% RSLogix 500 project ALSAFE.RSS, saved by version 8.10.00.18 %
PROJECT "ALSAFE"    % processor: SLC 500, 1747-L542 %

PROGRAM FILES
  LAD 2   73 rungs
  LAD 3   98 rungs
  LAD 4   40 rungs
  LAD 5   5 rungs
  LAD 6   89 rungs
  LAD 9   48 rungs
  LAD 10   101 rungs
  LAD 11   76 rungs
  LAD 15   61 rungs
  LAD 16   10 rungs
  LAD 17   20 rungs
  LAD 21   5 rungs
  LAD 22   77 rungs
  LAD 25   112 rungs
  LAD 26   32 rungs
  LAD 27   42 rungs
  LAD 30   28 rungs
  LAD 31   116 rungs
  LAD 32   20 rungs
  LAD 40   35 rungs
  LAD 50   183 rungs
  LAD 51   113 rungs
  LAD 52   5 rungs
  LAD 53   5 rungs
  LAD 71   9 rungs
  LAD 75   15 rungs
  LAD 76   23 rungs
  LAD 77   4 rungs
  LAD 78   4 rungs
  LAD 80   11 rungs

DATA FILES
  O0 OUTPUT  20 elements
  I1 INPUT  19 elements
  S2 STATUS  164 elements
  B3 BINARY  68 elements
  T4 TIMER  32 elements
  C5 COUNTER  2 elements
  R6 CONTROL  12 elements
  N7 INTEGER  131 elements
  F8 FLOAT  15 elements
  N9   25 elements
  B10   110 elements
  B11   63 elements
  T13   10 elements
  B15   1 elements
  B16   20 elements
  B17   28 elements
  T21   65 elements
  B22   11 elements
  B23   4 elements
  N25   210 elements
  B29   12 elements
  T31   40 elements
  N32   14 elements
  N40   60 elements
  N41   60 elements
  N42   120 elements
  B49   2 elements
  N50   54 elements
  N51   210 elements
  N52   18 elements
  B53   100 elements
  N54   31 elements
  N60   54 elements
  N75   250 elements
  N76   100 elements
  N90   5 elements
  N91   250 elements
  N92   250 elements
  N100   101 elements
  N104   12 elements
  N105   102 elements
  N106   1 elements
  N107   27 elements
  N108   12 elements
  N109   31 elements
  N111   214 elements

LADDER 2
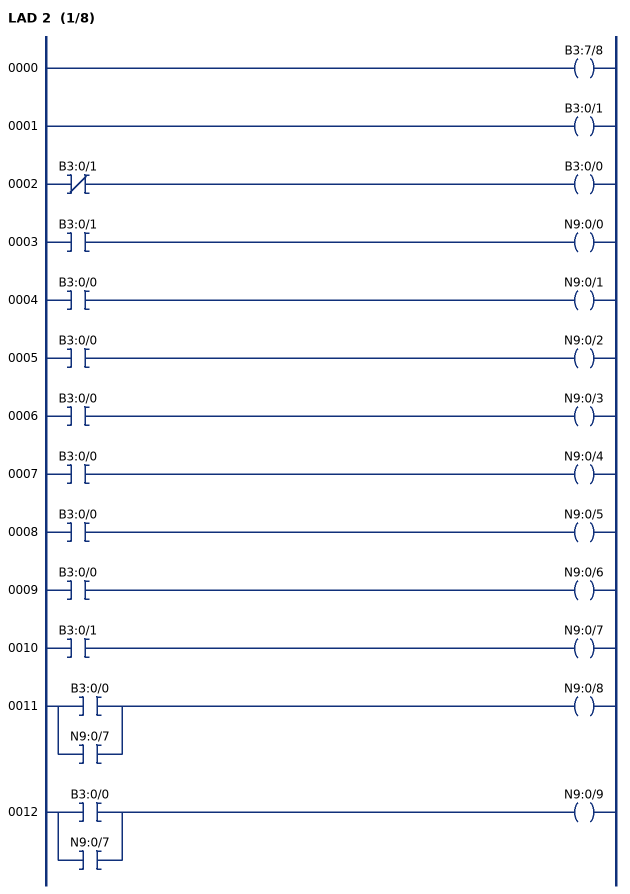
% Rung: 0 %
SOR OTE B3:7/8 EOR
% Rung: 1 %
SOR OTE B3:0/1 EOR
% Rung: 2 %
SOR XIO B3:0/1 OTE B3:0/0 EOR
% Rung: 3 %
SOR XIC B3:0/1 OTE N9:0/0 EOR
% Rung: 4 %
SOR XIC B3:0/0 OTE N9:0/1 EOR
% Rung: 5 %
SOR XIC B3:0/0 OTE N9:0/2 EOR
% Rung: 6 %
SOR XIC B3:0/0 OTE N9:0/3 EOR
% Rung: 7 %
SOR XIC B3:0/0 OTE N9:0/4 EOR
% Rung: 8 %
SOR XIC B3:0/0 OTE N9:0/5 EOR
% Rung: 9 %
SOR XIC B3:0/0 OTE N9:0/6 EOR
% Rung: 10 %
SOR XIC B3:0/1 OTE N9:0/7 EOR
% Rung: 11 %
SOR BST XIC B3:0/0 NXB XIC N9:0/7 BND OTE N9:0/8 EOR
% Rung: 12 %
SOR BST XIC B3:0/0 NXB XIC N9:0/7 BND OTE N9:0/9 EOR

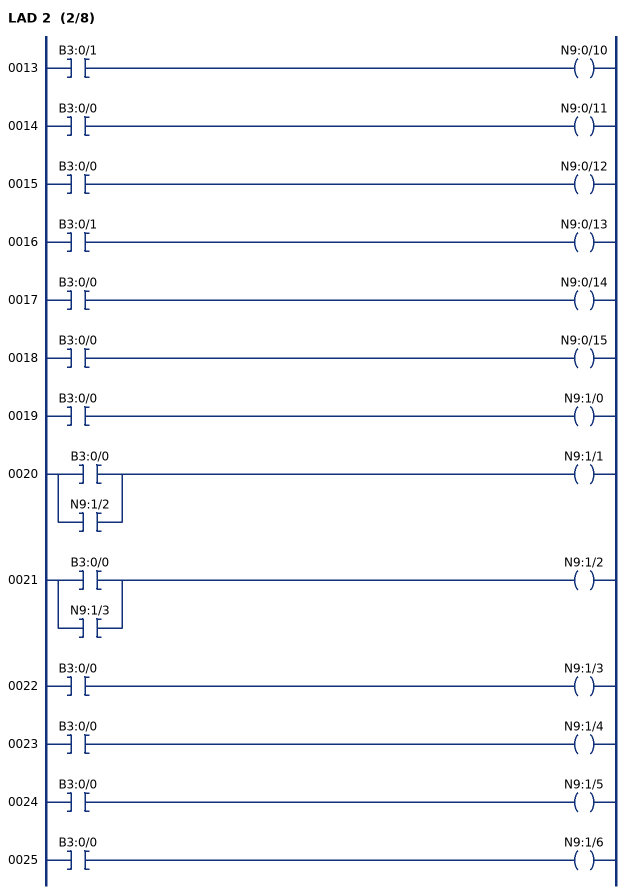
% Rung: 13 %
SOR XIC B3:0/1 OTE N9:0/10 EOR
% Rung: 14 %
SOR XIC B3:0/0 OTE N9:0/11 EOR
% Rung: 15 %
SOR XIC B3:0/0 OTE N9:0/12 EOR
% Rung: 16 %
SOR XIC B3:0/1 OTE N9:0/13 EOR
% Rung: 17 %
SOR XIC B3:0/0 OTE N9:0/14 EOR
% Rung: 18 %
SOR XIC B3:0/0 OTE N9:0/15 EOR
% Rung: 19 %
SOR XIC B3:0/0 OTE N9:1/0 EOR
% Rung: 20 %
SOR BST XIC B3:0/0 NXB XIC N9:1/2 BND OTE N9:1/1 EOR
% Rung: 21 %
SOR BST XIC B3:0/0 NXB XIC N9:1/3 BND OTE N9:1/2 EOR
% Rung: 22 %
SOR XIC B3:0/0 OTE N9:1/3 EOR
% Rung: 23 %
SOR XIC B3:0/0 OTE N9:1/4 EOR
% Rung: 24 %
SOR XIC B3:0/0 OTE N9:1/5 EOR
% Rung: 25 %
SOR XIC B3:0/0 OTE N9:1/6 EOR

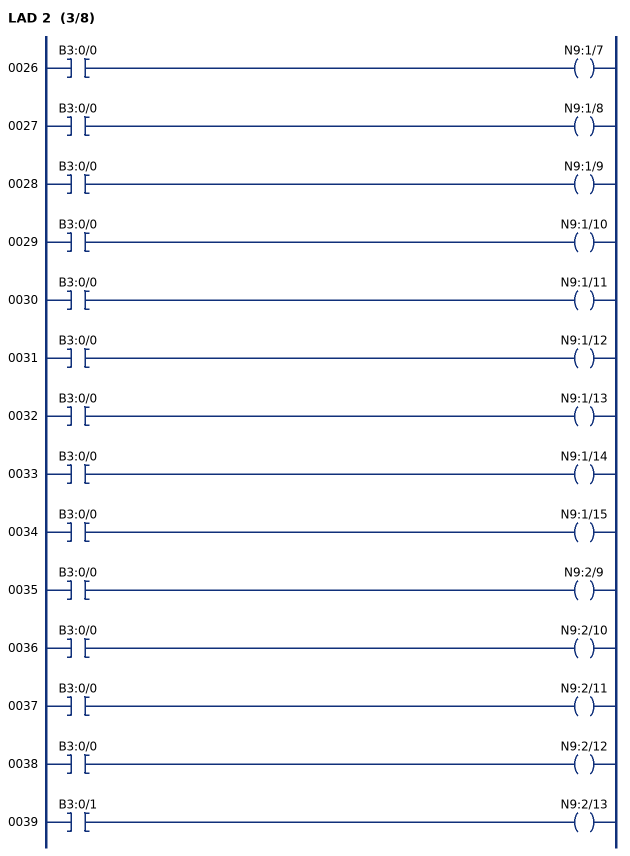
% Rung: 26 %
SOR XIC B3:0/0 OTE N9:1/7 EOR
% Rung: 27 %
SOR XIC B3:0/0 OTE N9:1/8 EOR
% Rung: 28 %
SOR XIC B3:0/0 OTE N9:1/9 EOR
% Rung: 29 %
SOR XIC B3:0/0 OTE N9:1/10 EOR
% Rung: 30 %
SOR XIC B3:0/0 OTE N9:1/11 EOR
% Rung: 31 %
SOR XIC B3:0/0 OTE N9:1/12 EOR
% Rung: 32 %
SOR XIC B3:0/0 OTE N9:1/13 EOR
% Rung: 33 %
SOR XIC B3:0/0 OTE N9:1/14 EOR
% Rung: 34 %
SOR XIC B3:0/0 OTE N9:1/15 EOR
% Rung: 35 %
SOR XIC B3:0/0 OTE N9:2/9 EOR
% Rung: 36 %
SOR XIC B3:0/0 OTE N9:2/10 EOR
% Rung: 37 %
SOR XIC B3:0/0 OTE N9:2/11 EOR
% Rung: 38 %
SOR XIC B3:0/0 OTE N9:2/12 EOR
% Rung: 39 %
SOR XIC B3:0/1 OTE N9:2/13 EOR

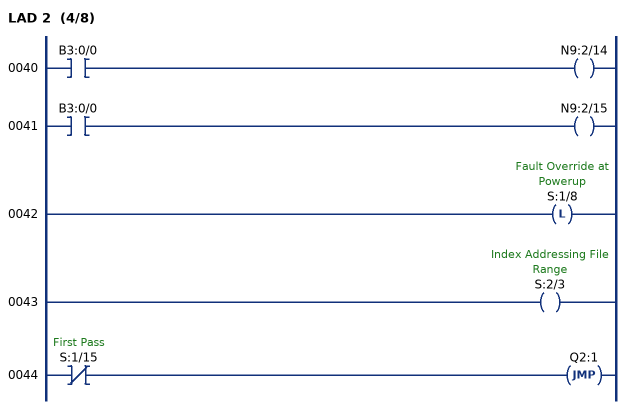
% Rung: 40 %
SOR XIC B3:0/0 OTE N9:2/14 EOR
% Rung: 41 %
SOR XIC B3:0/0 OTE N9:2/15 EOR
% Rung: 42 %
SOR OTL S:1/8 EOR
%   S:1/8  "Fault Override at Powerup" %
% Rung: 43 %
SOR OTE S:2/3 EOR
%   S:2/3  "Index Addressing File Range" %
% Rung: 44 %
SOR XIO S:1/15 JMP Q2:1 EOR
%   S:1/15  "First Pass" %

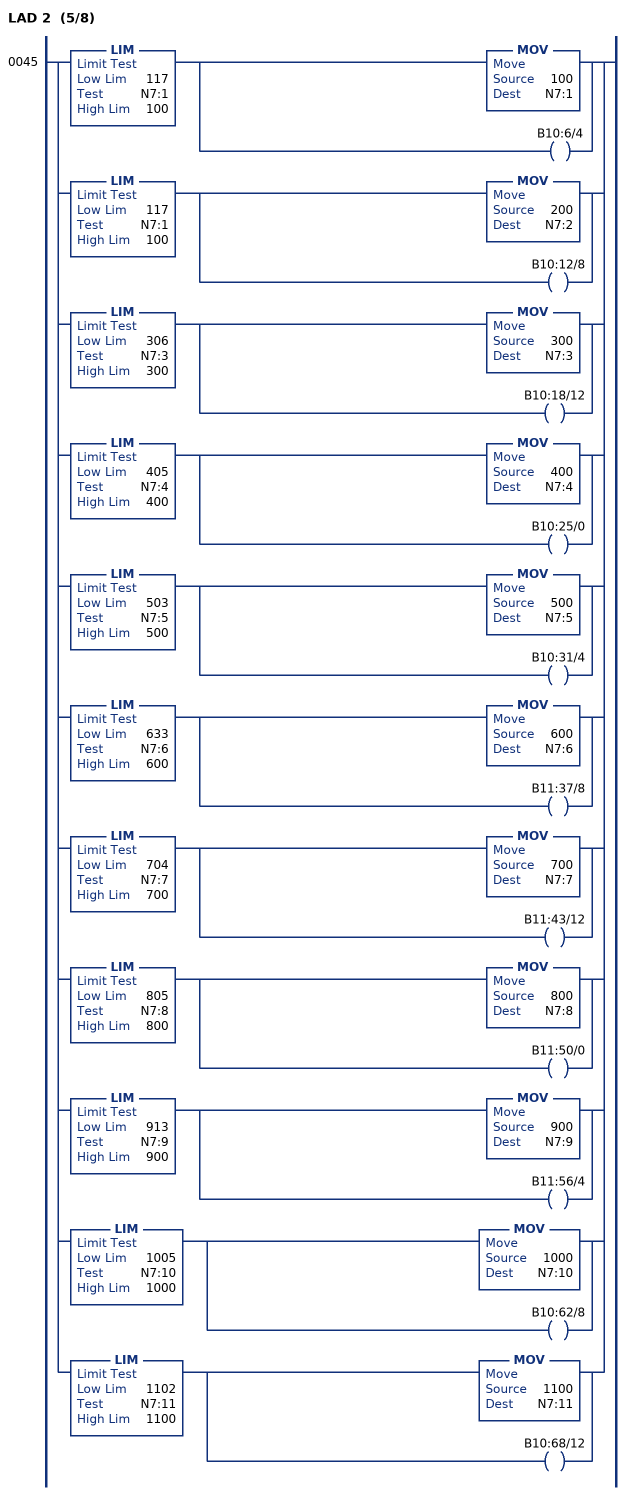
% Rung: 45 %
SOR BST LIM 117 N7:1 100 BST MOV 100 N7:1 NXB OTE B10:6/4 BND NXB LIM 117 N7:1 100 BST MOV 200 N7:2 NXB OTE B10:12/8 BND NXB LIM 306 N7:3 300 BST MOV 300 N7:3 NXB OTE B10:18/12 BND NXB LIM 405 N7:4 400 BST MOV 400 N7:4 NXB OTE B10:25/0 BND NXB LIM 503 N7:5 500 BST MOV 500 N7:5 NXB OTE B10:31/4 BND NXB LIM 633 N7:6 600 BST MOV 600 N7:6 NXB OTE B11:37/8 BND NXB LIM 704 N7:7 700 BST MOV 700 N7:7 NXB OTE B11:43/12 BND NXB LIM 805 N7:8 800 BST MOV 800 N7:8 NXB OTE B11:50/0 BND NXB LIM 913 N7:9 900 BST MOV 900 N7:9 NXB OTE B11:56/4 BND NXB LIM 1005 N7:10 1000 BST MOV 1000 N7:10 NXB OTE B10:62/8 BND NXB LIM 1102 N7:11 1100 BST MOV 1100 N7:11 NXB OTE B10:68/12 BND BND EOR

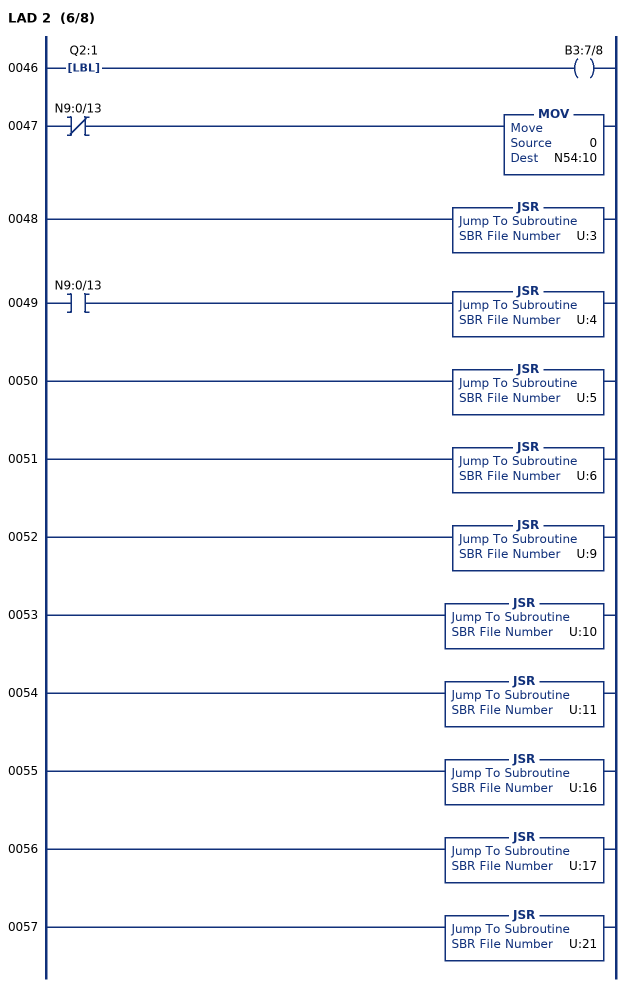
% Rung: 46 %
SOR LBL Q2:1 OTE B3:7/8 EOR
% Rung: 47 %
SOR XIO N9:0/13 MOV 0 N54:10 EOR
% Rung: 48 %
SOR JSR U:3 EOR
% Rung: 49 %
SOR XIC N9:0/13 JSR U:4 EOR
% Rung: 50 %
SOR JSR U:5 EOR
% Rung: 51 %
SOR JSR U:6 EOR
% Rung: 52 %
SOR JSR U:9 EOR
% Rung: 53 %
SOR JSR U:10 EOR
% Rung: 54 %
SOR JSR U:11 EOR
% Rung: 55 %
SOR JSR U:16 EOR
% Rung: 56 %
SOR JSR U:17 EOR
% Rung: 57 %
SOR JSR U:21 EOR

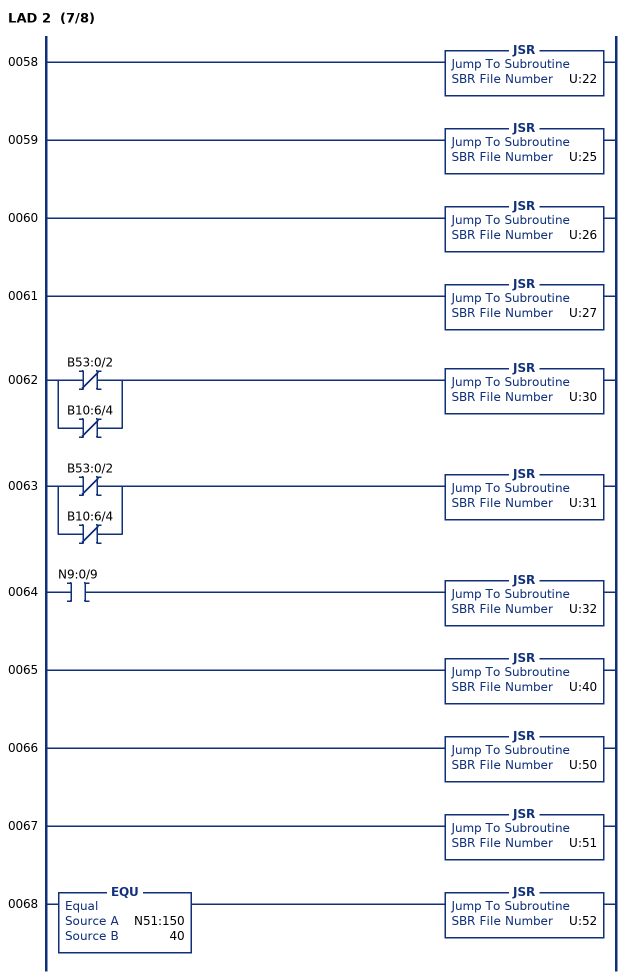
% Rung: 58 %
SOR JSR U:22 EOR
% Rung: 59 %
SOR JSR U:25 EOR
% Rung: 60 %
SOR JSR U:26 EOR
% Rung: 61 %
SOR JSR U:27 EOR
% Rung: 62 %
SOR BST XIO B53:0/2 NXB XIO B10:6/4 BND JSR U:30 EOR
% Rung: 63 %
SOR BST XIO B53:0/2 NXB XIO B10:6/4 BND JSR U:31 EOR
% Rung: 64 %
SOR XIC N9:0/9 JSR U:32 EOR
% Rung: 65 %
SOR JSR U:40 EOR
% Rung: 66 %
SOR JSR U:50 EOR
% Rung: 67 %
SOR JSR U:51 EOR
% Rung: 68 %
SOR EQU N51:150 40 JSR U:52 EOR

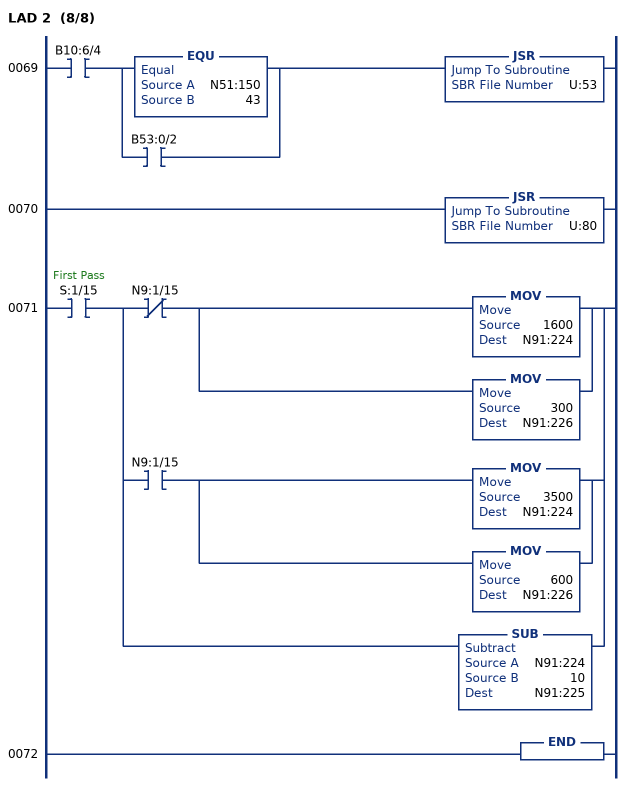
% Rung: 69 %
SOR XIC B10:6/4 BST EQU N51:150 43 NXB XIC B53:0/2 BND JSR U:53 EOR
% Rung: 70 %
SOR JSR U:80 EOR
% Rung: 71 %
SOR XIC S:1/15 BST XIO N9:1/15 BST MOV 1600 N91:224 NXB MOV 300 N91:226 BND NXB XIC N9:1/15 BST MOV 3500 N91:224 NXB MOV 600 N91:226 BND NXB SUB N91:224 10 N91:225 BND EOR
%   S:1/15  "First Pass" %
% Rung: 72 %
SOR END EOR

LADDER 3
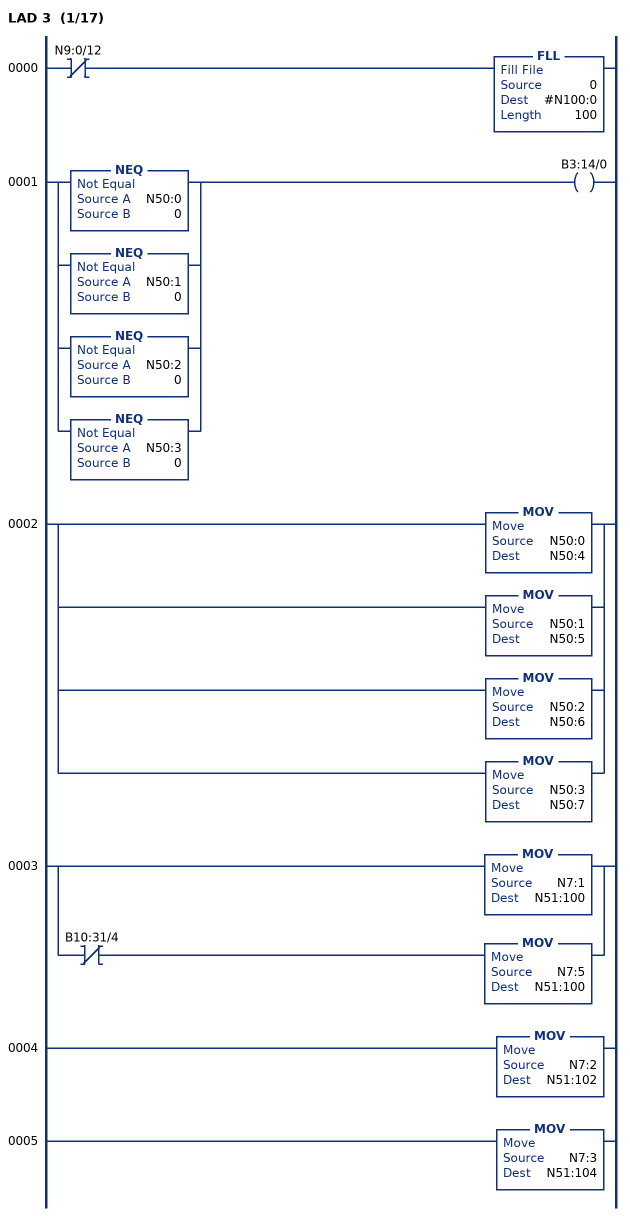
% Rung: 0 %
SOR XIO N9:0/12 FLL 0 #N100:0 100 EOR
% Rung: 1 %
SOR BST NEQ N50:0 0 NXB NEQ N50:1 0 NXB NEQ N50:2 0 NXB NEQ N50:3 0 BND OTE B3:14/0 EOR
% Rung: 2 %
SOR BST MOV N50:0 N50:4 NXB MOV N50:1 N50:5 NXB MOV N50:2 N50:6 NXB MOV N50:3 N50:7 BND EOR
% Rung: 3 %
SOR BST MOV N7:1 N51:100 NXB XIO B10:31/4 MOV N7:5 N51:100 BND EOR
% Rung: 4 %
SOR MOV N7:2 N51:102 EOR
% Rung: 5 %
SOR MOV N7:3 N51:104 EOR

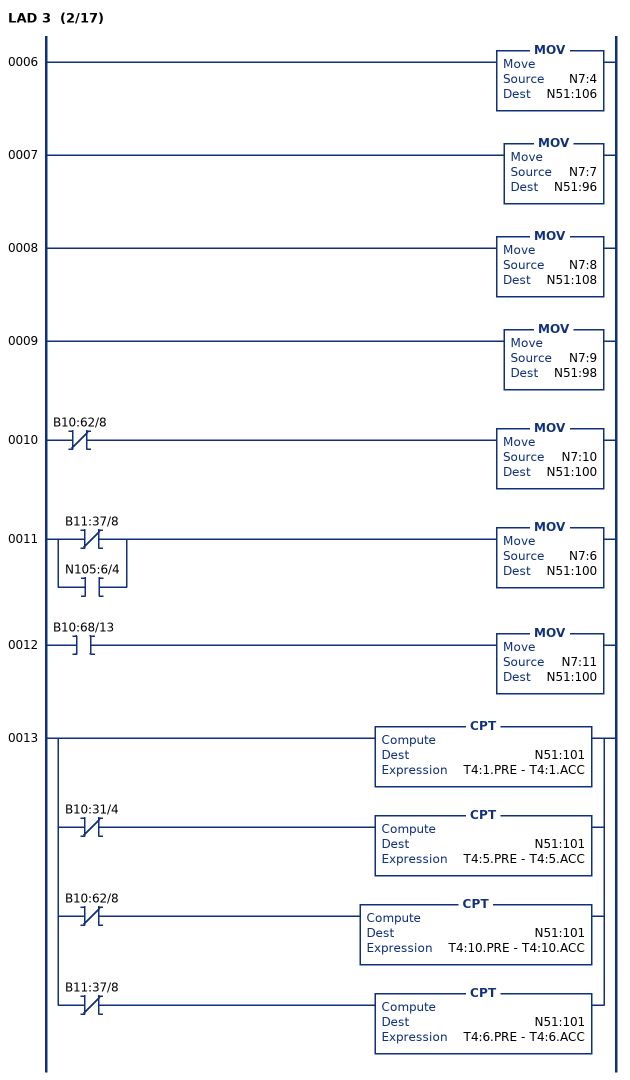
% Rung: 6 %
SOR MOV N7:4 N51:106 EOR
% Rung: 7 %
SOR MOV N7:7 N51:96 EOR
% Rung: 8 %
SOR MOV N7:8 N51:108 EOR
% Rung: 9 %
SOR MOV N7:9 N51:98 EOR
% Rung: 10 %
SOR XIO B10:62/8 MOV N7:10 N51:100 EOR
% Rung: 11 %
SOR BST XIO B11:37/8 NXB XIC N105:6/4 BND MOV N7:6 N51:100 EOR
% Rung: 12 %
SOR XIC B10:68/13 MOV N7:11 N51:100 EOR
% Rung: 13 %
SOR BST CPT N51:101 " T4:1.PRE - T4:1.ACC " NXB XIO B10:31/4 CPT N51:101 " T4:5.PRE - T4:5.ACC " NXB XIO B10:62/8 CPT N51:101 " T4:10.PRE - T4:10.ACC " NXB XIO B11:37/8 CPT N51:101 " T4:6.PRE - T4:6.ACC " BND EOR

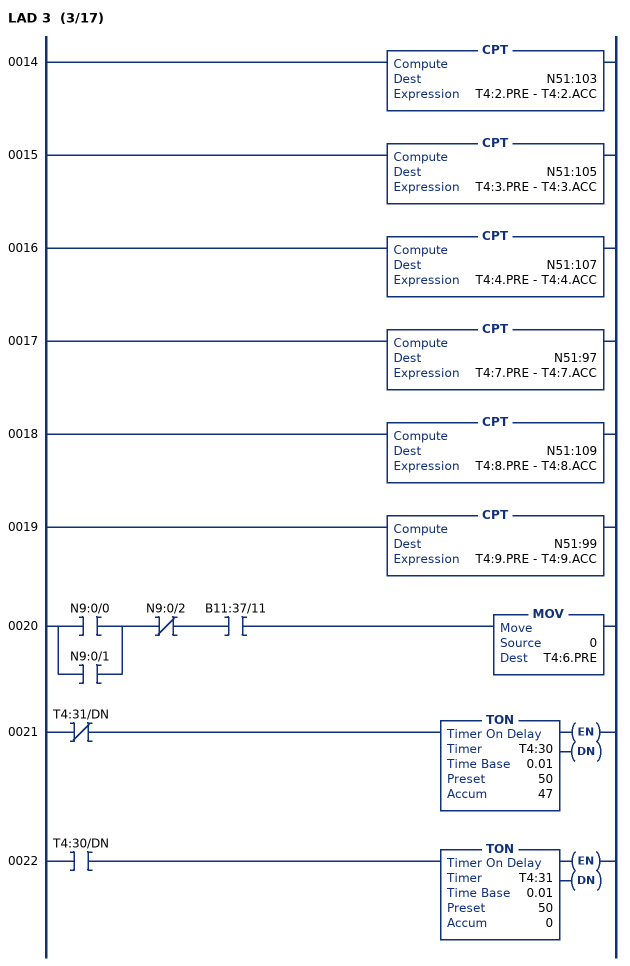
% Rung: 14 %
SOR CPT N51:103 " T4:2.PRE - T4:2.ACC " EOR
% Rung: 15 %
SOR CPT N51:105 " T4:3.PRE - T4:3.ACC " EOR
% Rung: 16 %
SOR CPT N51:107 " T4:4.PRE - T4:4.ACC " EOR
% Rung: 17 %
SOR CPT N51:97 " T4:7.PRE - T4:7.ACC " EOR
% Rung: 18 %
SOR CPT N51:109 " T4:8.PRE - T4:8.ACC " EOR
% Rung: 19 %
SOR CPT N51:99 " T4:9.PRE - T4:9.ACC " EOR
% Rung: 20 %
SOR BST XIC N9:0/0 NXB XIC N9:0/1 BND XIO N9:0/2 XIC B11:37/11 MOV 0 T4:6.PRE EOR
% Rung: 21 %
SOR XIO T4:31/DN TON T4:30 0.01 50 47 EOR
% Rung: 22 %
SOR XIC T4:30/DN TON T4:31 0.01 50 0 EOR

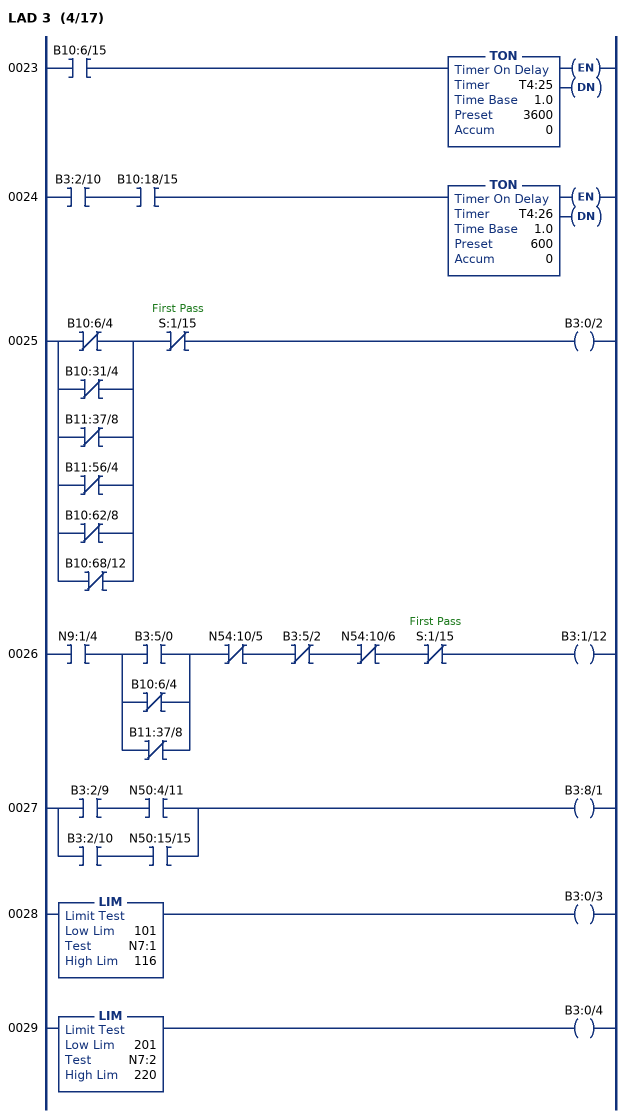
% Rung: 23 %
SOR XIC B10:6/15 TON T4:25 1.0 3600 0 EOR
% Rung: 24 %
SOR XIC B3:2/10 XIC B10:18/15 TON T4:26 1.0 600 0 EOR
% Rung: 25 %
SOR BST XIO B10:6/4 NXB XIO B10:31/4 NXB XIO B11:37/8 NXB XIO B11:56/4 NXB XIO B10:62/8 NXB XIO B10:68/12 BND XIO S:1/15 OTE B3:0/2 EOR
%   S:1/15  "First Pass" %
% Rung: 26 %
SOR XIC N9:1/4 BST XIC B3:5/0 NXB XIO B10:6/4 NXB XIO B11:37/8 BND XIO N54:10/5 XIO B3:5/2 XIO N54:10/6 XIO S:1/15 OTE B3:1/12 EOR
%   S:1/15  "First Pass" %
% Rung: 27 %
SOR BST XIC B3:2/9 XIC N50:4/11 NXB XIC B3:2/10 XIC N50:15/15 BND OTE B3:8/1 EOR
% Rung: 28 %
SOR LIM 101 N7:1 116 OTE B3:0/3 EOR
% Rung: 29 %
SOR LIM 201 N7:2 220 OTE B3:0/4 EOR

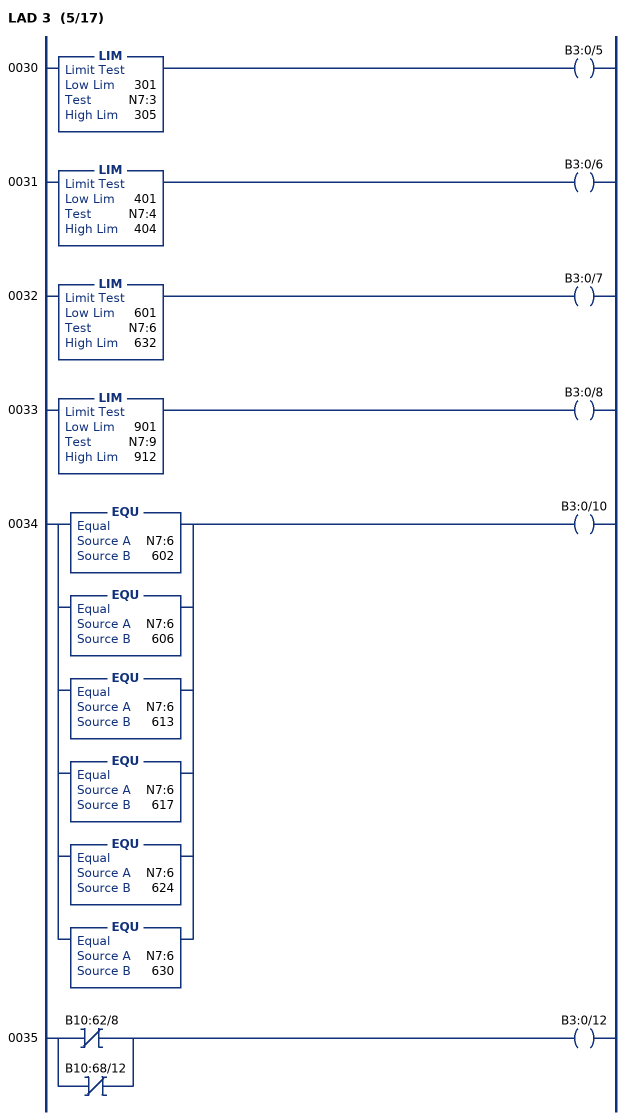
% Rung: 30 %
SOR LIM 301 N7:3 305 OTE B3:0/5 EOR
% Rung: 31 %
SOR LIM 401 N7:4 404 OTE B3:0/6 EOR
% Rung: 32 %
SOR LIM 601 N7:6 632 OTE B3:0/7 EOR
% Rung: 33 %
SOR LIM 901 N7:9 912 OTE B3:0/8 EOR
% Rung: 34 %
SOR BST EQU N7:6 602 NXB EQU N7:6 606 NXB EQU N7:6 613 NXB EQU N7:6 617 NXB EQU N7:6 624 NXB EQU N7:6 630 BND OTE B3:0/10 EOR
% Rung: 35 %
SOR BST XIO B10:62/8 NXB XIO B10:68/12 BND OTE B3:0/12 EOR

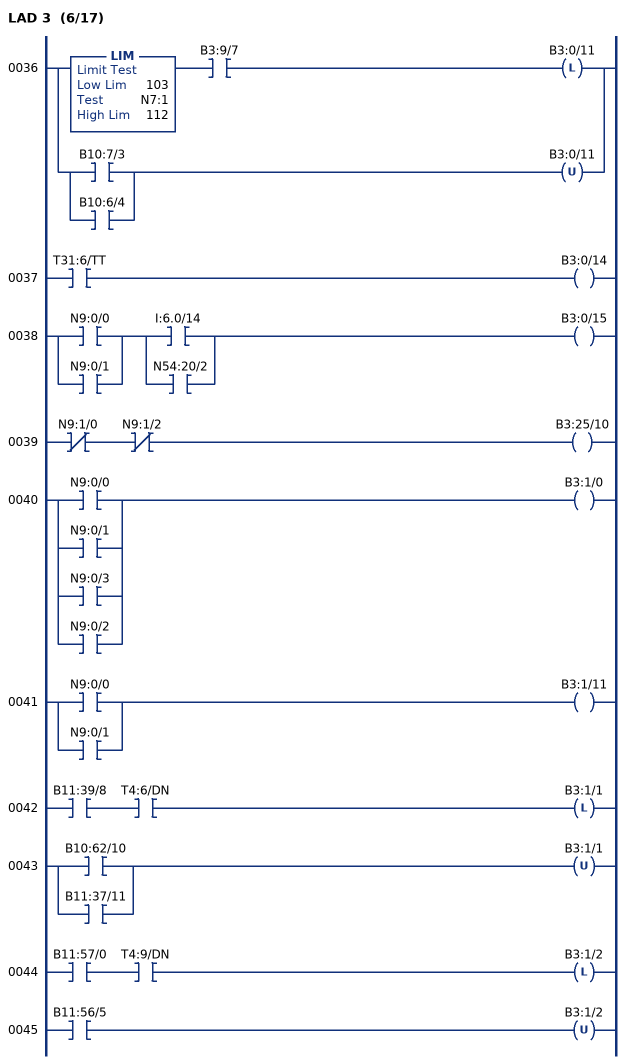
% Rung: 36 %
SOR BST LIM 103 N7:1 112 XIC B3:9/7 OTL B3:0/11 NXB BST XIC B10:7/3 NXB XIC B10:6/4 BND OTU B3:0/11 BND EOR
% Rung: 37 %
SOR XIC T31:6/TT OTE B3:0/14 EOR
% Rung: 38 %
SOR BST XIC N9:0/0 NXB XIC N9:0/1 BND BST XIC I:6.0/14 NXB XIC N54:20/2 BND OTE B3:0/15 EOR
% Rung: 39 %
SOR XIO N9:1/0 XIO N9:1/2 OTE B3:25/10 EOR
% Rung: 40 %
SOR BST XIC N9:0/0 NXB XIC N9:0/1 NXB XIC N9:0/3 NXB XIC N9:0/2 BND OTE B3:1/0 EOR
% Rung: 41 %
SOR BST XIC N9:0/0 NXB XIC N9:0/1 BND OTE B3:1/11 EOR
% Rung: 42 %
SOR XIC B11:39/8 XIC T4:6/DN OTL B3:1/1 EOR
% Rung: 43 %
SOR BST XIC B10:62/10 NXB XIC B11:37/11 BND OTU B3:1/1 EOR
% Rung: 44 %
SOR XIC B11:57/0 XIC T4:9/DN OTL B3:1/2 EOR
% Rung: 45 %
SOR XIC B11:56/5 OTU B3:1/2 EOR

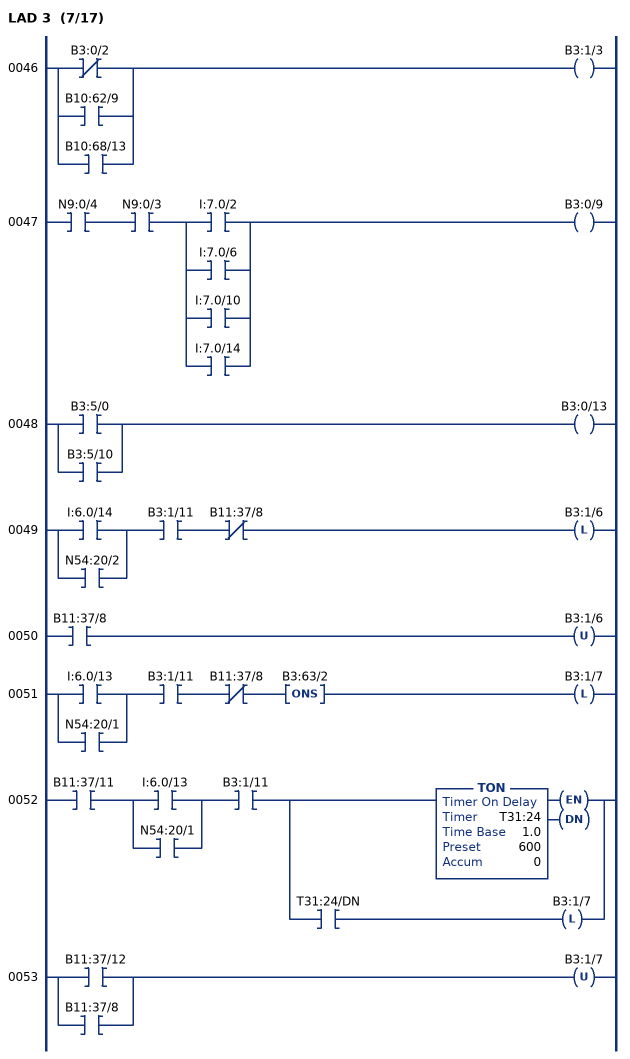
% Rung: 46 %
SOR BST XIO B3:0/2 NXB XIC B10:62/9 NXB XIC B10:68/13 BND OTE B3:1/3 EOR
% Rung: 47 %
SOR XIC N9:0/4 XIC N9:0/3 BST XIC I:7.0/2 NXB XIC I:7.0/6 NXB XIC I:7.0/10 NXB XIC I:7.0/14 BND OTE B3:0/9 EOR
% Rung: 48 %
SOR BST XIC B3:5/0 NXB XIC B3:5/10 BND OTE B3:0/13 EOR
% Rung: 49 %
SOR BST XIC I:6.0/14 NXB XIC N54:20/2 BND XIC B3:1/11 XIO B11:37/8 OTL B3:1/6 EOR
% Rung: 50 %
SOR XIC B11:37/8 OTU B3:1/6 EOR
% Rung: 51 %
SOR BST XIC I:6.0/13 NXB XIC N54:20/1 BND XIC B3:1/11 XIO B11:37/8 OSR B3:63/2 OTL B3:1/7 EOR
% Rung: 52 %
SOR XIC B11:37/11 BST XIC I:6.0/13 NXB XIC N54:20/1 BND XIC B3:1/11 BST TON T31:24 1.0 600 0 NXB XIC T31:24/DN OTL B3:1/7 BND EOR
% Rung: 53 %
SOR BST XIC B11:37/12 NXB XIC B11:37/8 BND OTU B3:1/7 EOR

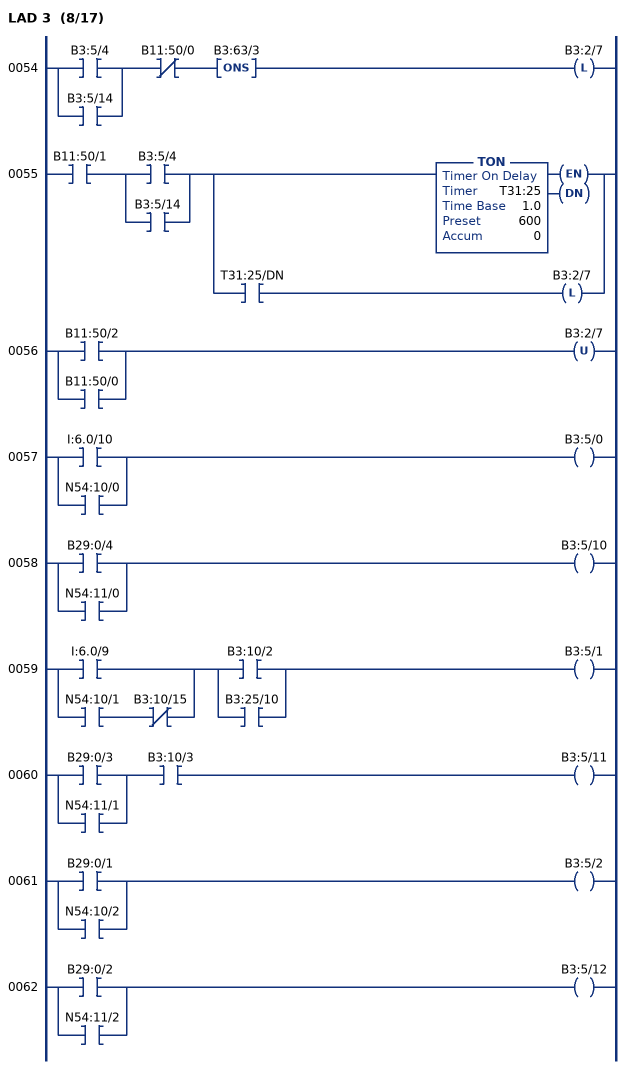
% Rung: 54 %
SOR BST XIC B3:5/4 NXB XIC B3:5/14 BND XIO B11:50/0 OSR B3:63/3 OTL B3:2/7 EOR
% Rung: 55 %
SOR XIC B11:50/1 BST XIC B3:5/4 NXB XIC B3:5/14 BND BST TON T31:25 1.0 600 0 NXB XIC T31:25/DN OTL B3:2/7 BND EOR
% Rung: 56 %
SOR BST XIC B11:50/2 NXB XIC B11:50/0 BND OTU B3:2/7 EOR
% Rung: 57 %
SOR BST XIC I:6.0/10 NXB XIC N54:10/0 BND OTE B3:5/0 EOR
% Rung: 58 %
SOR BST XIC B29:0/4 NXB XIC N54:11/0 BND OTE B3:5/10 EOR
% Rung: 59 %
SOR BST XIC I:6.0/9 NXB XIC N54:10/1 XIO B3:10/15 BND BST XIC B3:10/2 NXB XIC B3:25/10 BND OTE B3:5/1 EOR
% Rung: 60 %
SOR BST XIC B29:0/3 NXB XIC N54:11/1 BND XIC B3:10/3 OTE B3:5/11 EOR
% Rung: 61 %
SOR BST XIC B29:0/1 NXB XIC N54:10/2 BND OTE B3:5/2 EOR
% Rung: 62 %
SOR BST XIC B29:0/2 NXB XIC N54:11/2 BND OTE B3:5/12 EOR

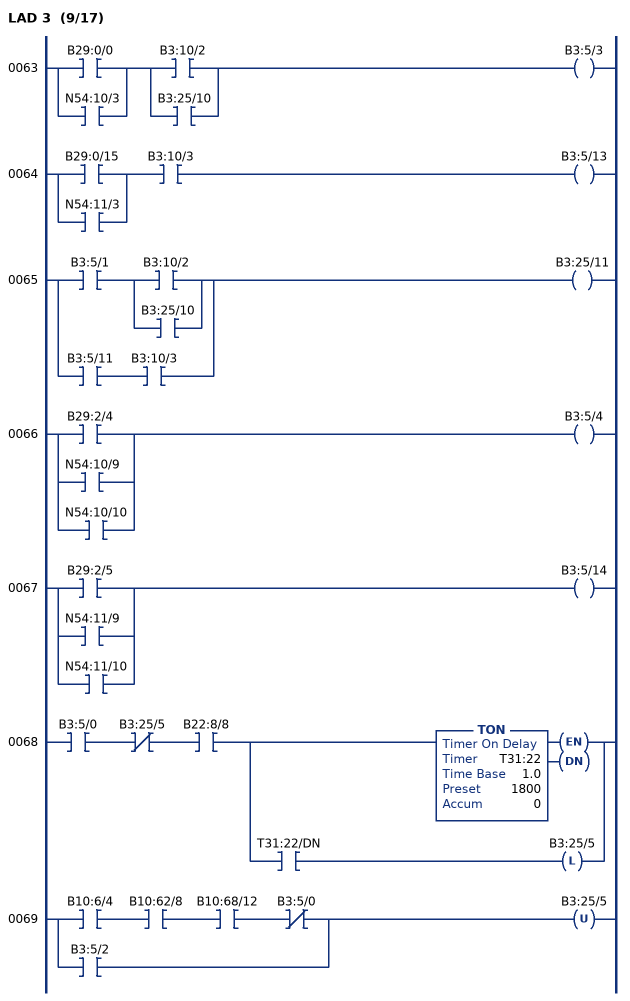
% Rung: 63 %
SOR BST XIC B29:0/0 NXB XIC N54:10/3 BND BST XIC B3:10/2 NXB XIC B3:25/10 BND OTE B3:5/3 EOR
% Rung: 64 %
SOR BST XIC B29:0/15 NXB XIC N54:11/3 BND XIC B3:10/3 OTE B3:5/13 EOR
% Rung: 65 %
SOR BST XIC B3:5/1 BST XIC B3:10/2 NXB XIC B3:25/10 BND NXB XIC B3:5/11 XIC B3:10/3 BND OTE B3:25/11 EOR
% Rung: 66 %
SOR BST XIC B29:2/4 NXB XIC N54:10/9 NXB XIC N54:10/10 BND OTE B3:5/4 EOR
% Rung: 67 %
SOR BST XIC B29:2/5 NXB XIC N54:11/9 NXB XIC N54:11/10 BND OTE B3:5/14 EOR
% Rung: 68 %
SOR XIC B3:5/0 XIO B3:25/5 XIC B22:8/8 BST TON T31:22 1.0 1800 0 NXB XIC T31:22/DN OTL B3:25/5 BND EOR
% Rung: 69 %
SOR BST XIC B10:6/4 XIC B10:62/8 XIC B10:68/12 XIO B3:5/0 NXB XIC B3:5/2 BND OTU B3:25/5 EOR

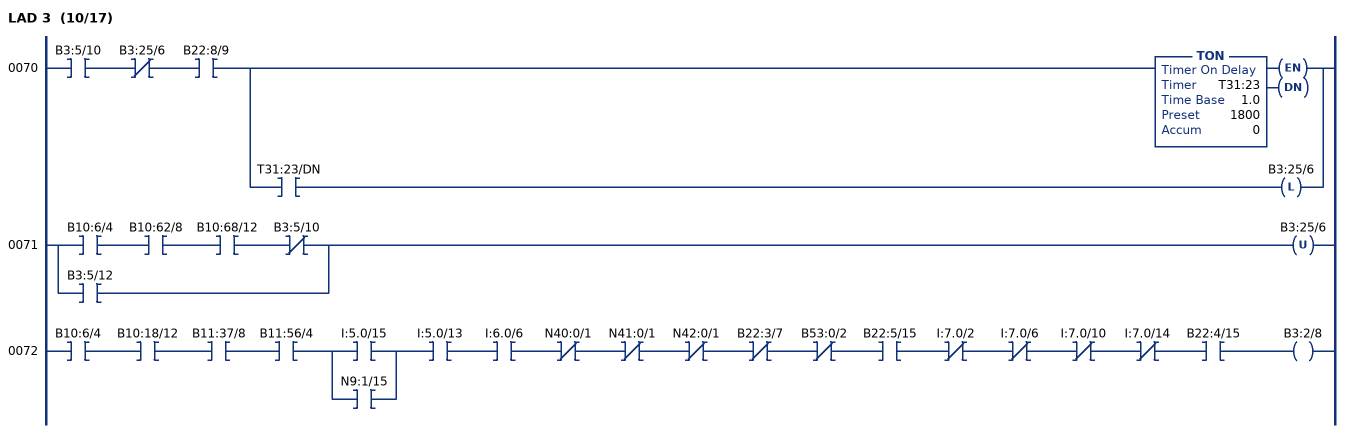
% Rung: 70 %
SOR XIC B3:5/10 XIO B3:25/6 XIC B22:8/9 BST TON T31:23 1.0 1800 0 NXB XIC T31:23/DN OTL B3:25/6 BND EOR
% Rung: 71 %
SOR BST XIC B10:6/4 XIC B10:62/8 XIC B10:68/12 XIO B3:5/10 NXB XIC B3:5/12 BND OTU B3:25/6 EOR
% Rung: 72 %
SOR XIC B10:6/4 XIC B10:18/12 XIC B11:37/8 XIC B11:56/4 BST XIC I:5.0/15 NXB XIC N9:1/15 BND XIC I:5.0/13 XIC I:6.0/6 XIO N40:0/1 XIO N41:0/1 XIO N42:0/1 XIO B22:3/7 XIO B53:0/2 XIC B22:5/15 XIO I:7.0/2 XIO I:7.0/6 XIO I:7.0/10 XIO I:7.0/14 XIC B22:4/15 OTE B3:2/8 EOR

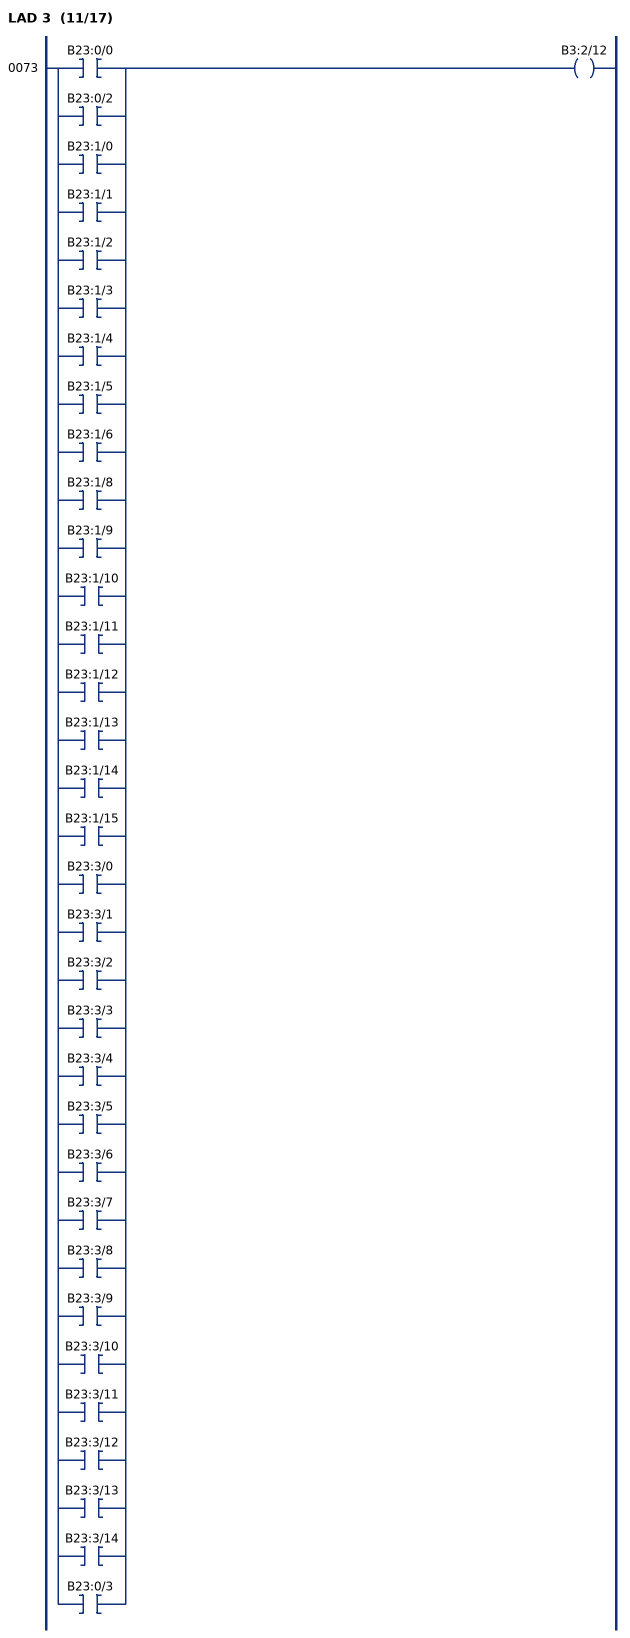
% Rung: 73 %
SOR BST XIC B23:0/0 NXB XIC B23:0/2 NXB XIC B23:1/0 NXB XIC B23:1/1 NXB XIC B23:1/2 NXB XIC B23:1/3 NXB XIC B23:1/4 NXB XIC B23:1/5 NXB XIC B23:1/6 NXB XIC B23:1/8 NXB XIC B23:1/9 NXB XIC B23:1/10 NXB XIC B23:1/11 NXB XIC B23:1/12 NXB XIC B23:1/13 NXB XIC B23:1/14 NXB XIC B23:1/15 NXB XIC B23:3/0 NXB XIC B23:3/1 NXB XIC B23:3/2 NXB XIC B23:3/3 NXB XIC B23:3/4 NXB XIC B23:3/5 NXB XIC B23:3/6 NXB XIC B23:3/7 NXB XIC B23:3/8 NXB XIC B23:3/9 NXB XIC B23:3/10 NXB XIC B23:3/11 NXB XIC B23:3/12 NXB XIC B23:3/13 NXB XIC B23:3/14 NXB XIC B23:0/3 BND OTE B3:2/12 EOR

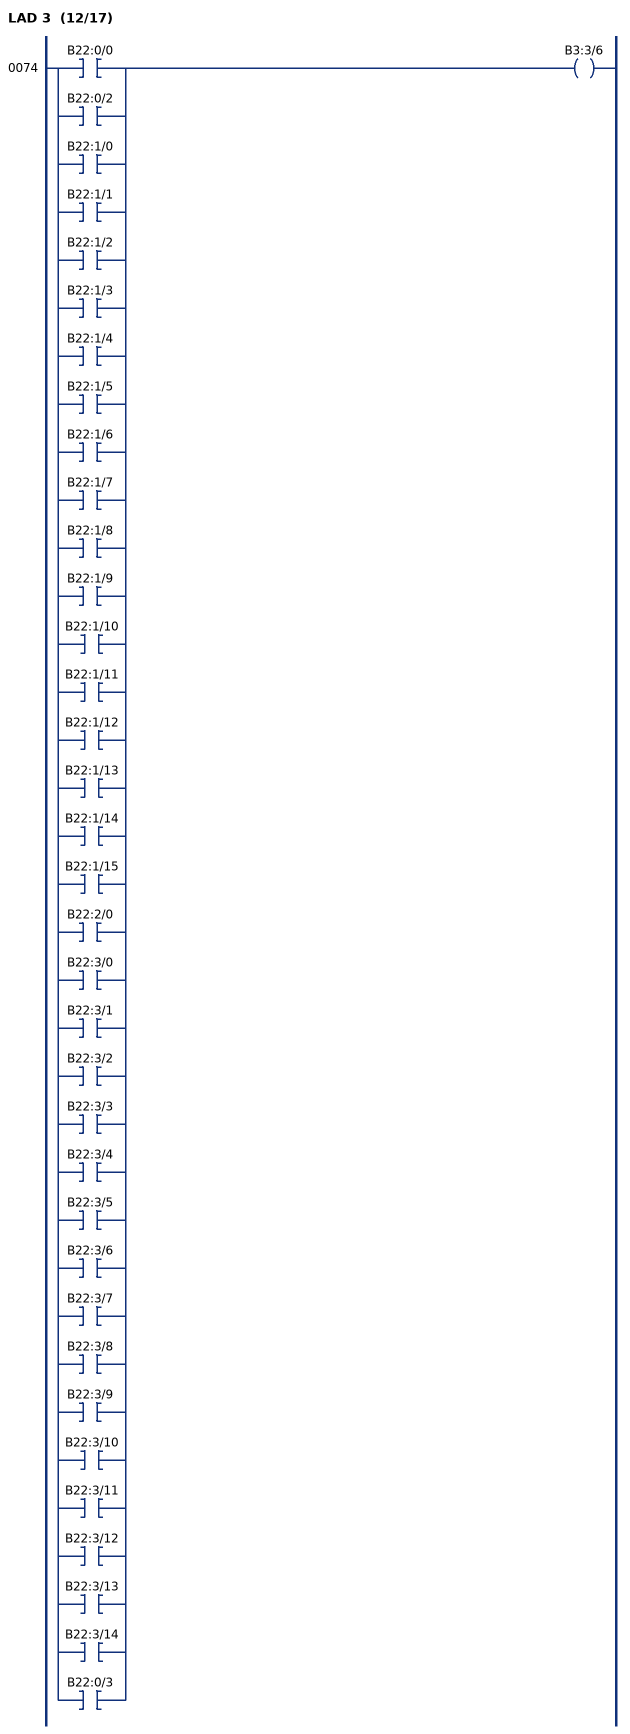
% Rung: 74 %
SOR BST XIC B22:0/0 NXB XIC B22:0/2 NXB XIC B22:1/0 NXB XIC B22:1/1 NXB XIC B22:1/2 NXB XIC B22:1/3 NXB XIC B22:1/4 NXB XIC B22:1/5 NXB XIC B22:1/6 NXB XIC B22:1/7 NXB XIC B22:1/8 NXB XIC B22:1/9 NXB XIC B22:1/10 NXB XIC B22:1/11 NXB XIC B22:1/12 NXB XIC B22:1/13 NXB XIC B22:1/14 NXB XIC B22:1/15 NXB XIC B22:2/0 NXB XIC B22:3/0 NXB XIC B22:3/1 NXB XIC B22:3/2 NXB XIC B22:3/3 NXB XIC B22:3/4 NXB XIC B22:3/5 NXB XIC B22:3/6 NXB XIC B22:3/7 NXB XIC B22:3/8 NXB XIC B22:3/9 NXB XIC B22:3/10 NXB XIC B22:3/11 NXB XIC B22:3/12 NXB XIC B22:3/13 NXB XIC B22:3/14 NXB XIC B22:0/3 BND OTE B3:3/6 EOR

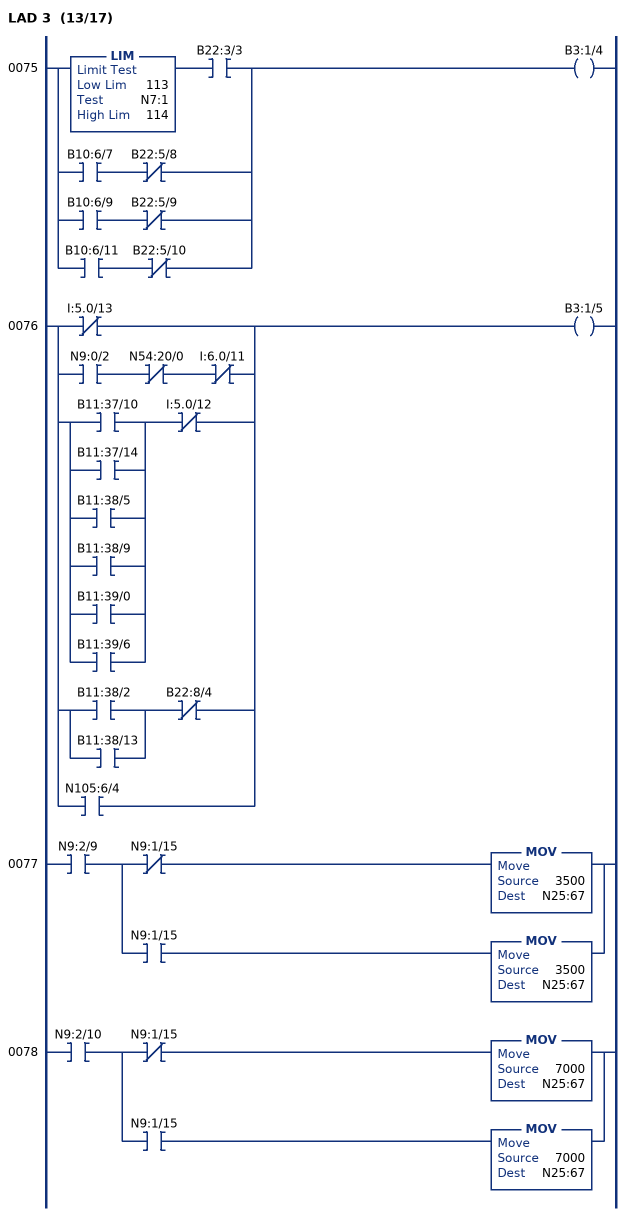
% Rung: 75 %
SOR BST LIM 113 N7:1 114 XIC B22:3/3 NXB XIC B10:6/7 XIO B22:5/8 NXB XIC B10:6/9 XIO B22:5/9 NXB XIC B10:6/11 XIO B22:5/10 BND OTE B3:1/4 EOR
% Rung: 76 %
SOR BST XIO I:5.0/13 NXB XIC N9:0/2 XIO N54:20/0 XIO I:6.0/11 NXB BST XIC B11:37/10 NXB XIC B11:37/14 NXB XIC B11:38/5 NXB XIC B11:38/9 NXB XIC B11:39/0 NXB XIC B11:39/6 BND XIO I:5.0/12 NXB BST XIC B11:38/2 NXB XIC B11:38/13 BND XIO B22:8/4 NXB XIC N105:6/4 BND OTE B3:1/5 EOR
% Rung: 77 %
SOR XIC N9:2/9 BST XIO N9:1/15 MOV 3500 N25:67 NXB XIC N9:1/15 MOV 3500 N25:67 BND EOR
% Rung: 78 %
SOR XIC N9:2/10 BST XIO N9:1/15 MOV 7000 N25:67 NXB XIC N9:1/15 MOV 7000 N25:67 BND EOR

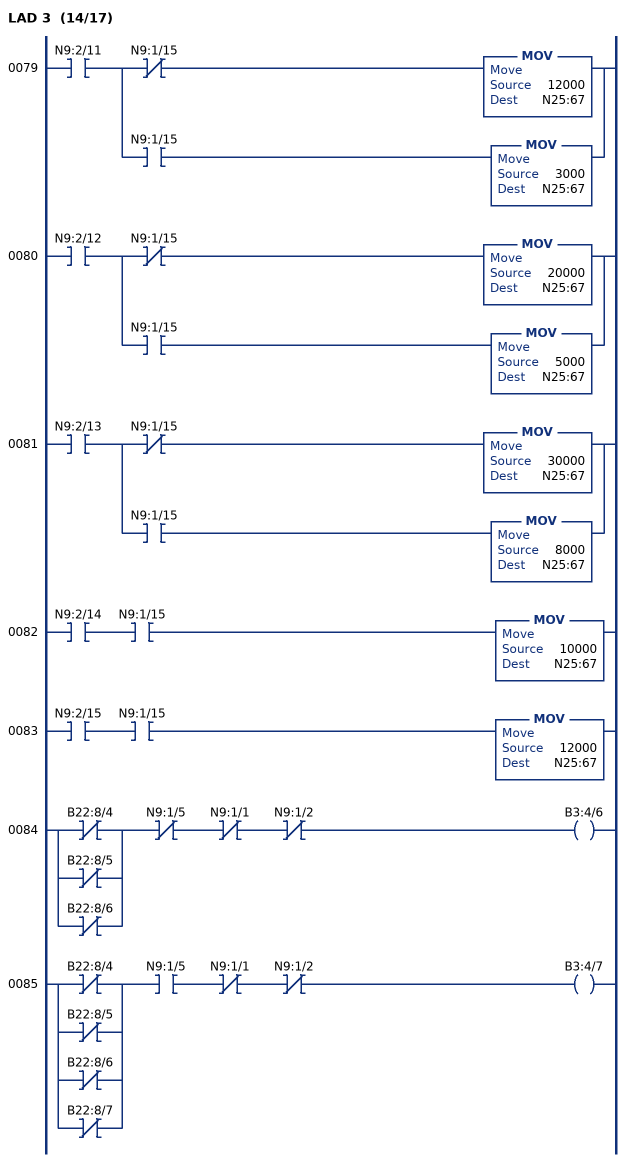
% Rung: 79 %
SOR XIC N9:2/11 BST XIO N9:1/15 MOV 12000 N25:67 NXB XIC N9:1/15 MOV 3000 N25:67 BND EOR
% Rung: 80 %
SOR XIC N9:2/12 BST XIO N9:1/15 MOV 20000 N25:67 NXB XIC N9:1/15 MOV 5000 N25:67 BND EOR
% Rung: 81 %
SOR XIC N9:2/13 BST XIO N9:1/15 MOV 30000 N25:67 NXB XIC N9:1/15 MOV 8000 N25:67 BND EOR
% Rung: 82 %
SOR XIC N9:2/14 XIC N9:1/15 MOV 10000 N25:67 EOR
% Rung: 83 %
SOR XIC N9:2/15 XIC N9:1/15 MOV 12000 N25:67 EOR
% Rung: 84 %
SOR BST XIO B22:8/4 NXB XIO B22:8/5 NXB XIO B22:8/6 BND XIO N9:1/5 XIO N9:1/1 XIO N9:1/2 OTE B3:4/6 EOR
% Rung: 85 %
SOR BST XIO B22:8/4 NXB XIO B22:8/5 NXB XIO B22:8/6 NXB XIO B22:8/7 BND XIC N9:1/5 XIO N9:1/1 XIO N9:1/2 OTE B3:4/7 EOR

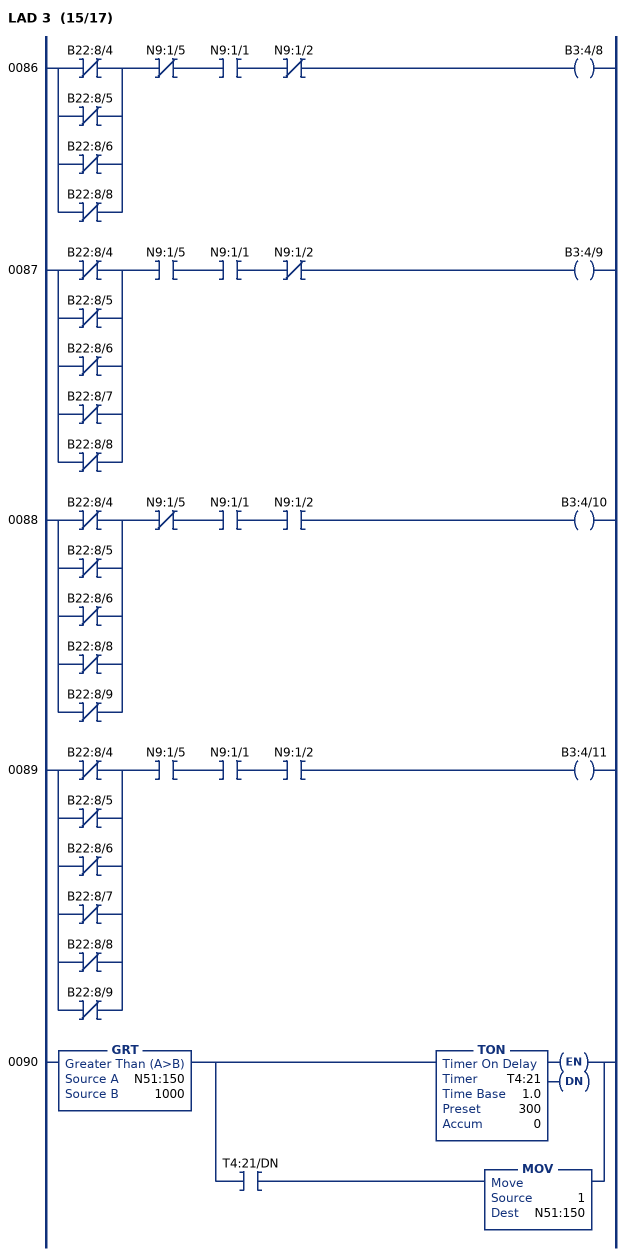
% Rung: 86 %
SOR BST XIO B22:8/4 NXB XIO B22:8/5 NXB XIO B22:8/6 NXB XIO B22:8/8 BND XIO N9:1/5 XIC N9:1/1 XIO N9:1/2 OTE B3:4/8 EOR
% Rung: 87 %
SOR BST XIO B22:8/4 NXB XIO B22:8/5 NXB XIO B22:8/6 NXB XIO B22:8/7 NXB XIO B22:8/8 BND XIC N9:1/5 XIC N9:1/1 XIO N9:1/2 OTE B3:4/9 EOR
% Rung: 88 %
SOR BST XIO B22:8/4 NXB XIO B22:8/5 NXB XIO B22:8/6 NXB XIO B22:8/8 NXB XIO B22:8/9 BND XIO N9:1/5 XIC N9:1/1 XIC N9:1/2 OTE B3:4/10 EOR
% Rung: 89 %
SOR BST XIO B22:8/4 NXB XIO B22:8/5 NXB XIO B22:8/6 NXB XIO B22:8/7 NXB XIO B22:8/8 NXB XIO B22:8/9 BND XIC N9:1/5 XIC N9:1/1 XIC N9:1/2 OTE B3:4/11 EOR
% Rung: 90 %
SOR GRT N51:150 1000 BST TON T4:21 1.0 300 0 NXB XIC T4:21/DN MOV 1 N51:150 BND EOR

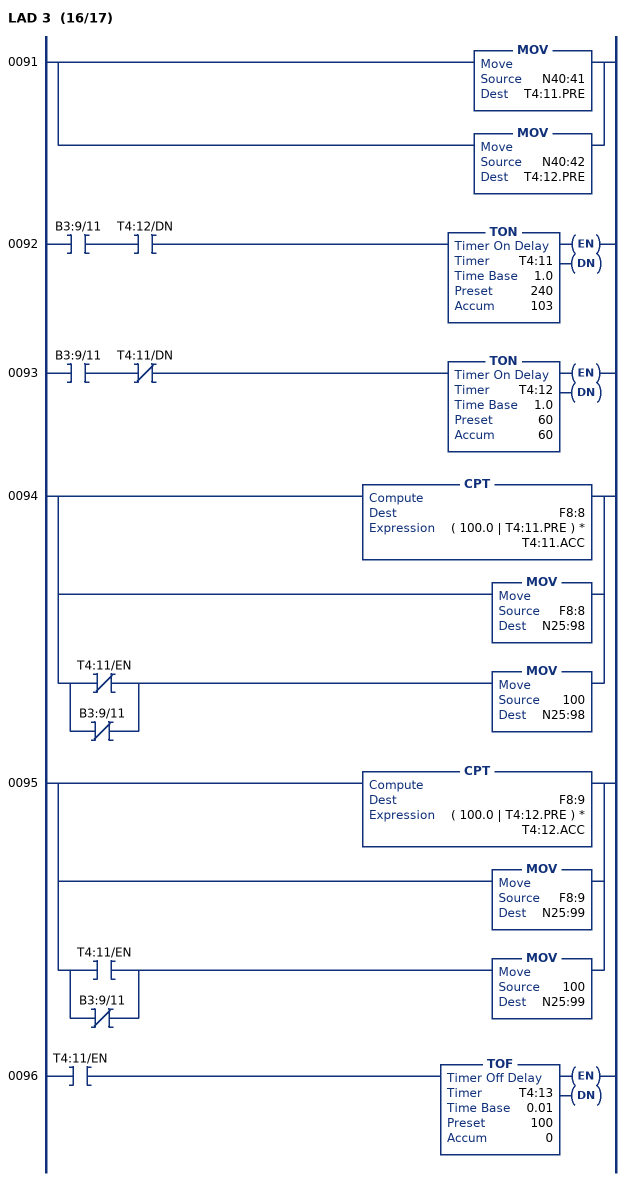
% Rung: 91 %
SOR BST MOV N40:41 T4:11.PRE NXB MOV N40:42 T4:12.PRE BND EOR
% Rung: 92 %
SOR XIC B3:9/11 XIC T4:12/DN TON T4:11 1.0 240 103 EOR
% Rung: 93 %
SOR XIC B3:9/11 XIO T4:11/DN TON T4:12 1.0 60 60 EOR
% Rung: 94 %
SOR BST CPT F8:8 " ( 100.0 | T4:11.PRE ) * T4:11.ACC " NXB MOV F8:8 N25:98 NXB BST XIO T4:11/EN NXB XIO B3:9/11 BND MOV 100 N25:98 BND EOR
% Rung: 95 %
SOR BST CPT F8:9 " ( 100.0 | T4:12.PRE ) * T4:12.ACC " NXB MOV F8:9 N25:99 NXB BST XIC T4:11/EN NXB XIO B3:9/11 BND MOV 100 N25:99 BND EOR
% Rung: 96 %
SOR XIC T4:11/EN TOF T4:13 0.01 100 0 EOR

